// TwinCAT 3 PLC project PersoneelsData
// ProgramVersion: 3.1.4024.0
// libraries:
//   StringUtils, * (System)
//   Tc2_Standard, * (Beckhoff Automation GmbH)
//   Tc2_System, * (Beckhoff Automation GmbH)
//   Tc3_Module, * (Beckhoff Automation GmbH)
// project tree:
//   DUTs/ Pers_data.TcDUT
//   / PlcTask.TcTTO
//   POUs/ FB_CheckString.TcPOU, MAIN.TcPOU
// (motion and I/O tree: see PLC project checkerfunctions)
// real-time tasks:
//   TASK PlcTask: cycle T#10ms, priority 20, ADS port 350
//   TASK PlcTask1: cycle T#10ms, priority 21, ADS port 351
//   TASK PlcTask2: cycle T#10ms, priority 22, ADS port 352
//   TASK PlcTask3: cycle T#10ms, priority 23, ADS port 353
//   TASK PlcTask4: cycle T#10ms, priority 24, ADS port 354
//   TASK PlcTask5: cycle T#10ms, priority 25, ADS port 355
//   TASK PlcTask6: cycle T#10ms, priority 26, ADS port 356
//   TASK PlcTask7: cycle T#10ms, priority 27, ADS port 357

CONFIGURATION PersoneelsData
    RESOURCE PLC ON TwinCAT3
        TASK PlcTask(INTERVAL := T#10ms, PRIORITY := 24);
        PROGRAM MAIN WITH PlcTask : MAIN;
    END_RESOURCE
END_CONFIGURATION

// ---- DUTs/Pers_data.TcDUT
TYPE Pers_data :
STRUCT
    Name : STRING[25];
    Firstname : STRING[25];
    Gender : STRING[10]; // 'Male' of 'Female'
    Age : INT;
    Address : STRING[55];
END_STRUCT
END_TYPE

// ---- POUs/MAIN.TcPOU
PROGRAM MAIN
VAR
    PersonnelArray : ARRAY [1..6] OF Pers_data := [
        (Name := 'Müller', Firstname := 'Peter', Gender := 'Male', Age := 32, Address := 'Postweg 34'),
        (Name := 'Fossen', Firstname := 'Jo', Gender := 'Male', Age := 20, Address := 'Broekstraat 45'),
        (Name := 'Maesen', Firstname := 'Stijn', Gender := 'Male', Age := 15, Address := 'Grote steenweg 8'),
        (Name := 'Poesmans', Firstname := 'Benny', Gender := 'Male', Age := 72, Address := 'Veldweg 1A'),
        (Name := 'Paque', Firstname := 'Stéphanie', Gender := 'Female', Age := 42, Address := 'Tongersesteenweg 456'),
        (Name := 'Dybek', Firstname := 'Isolde', Gender := 'Female', Age := 55, Address := 'Slagerijstraat 6')
    ];
	
	myData : Pers_data; // Vul myData met de gewenste waarden
    searchString : STRING := 'Stijn'; // De te zoeken string
    result : BOOL; // Resultaat van de zoekactie
    checkStringFB : FB_CheckString; // Aanmaken van de FB-instance
END_VAR

// NOG NIET OPGELOST!!!


// Vul myData met gegevens

checkStringFB.data := myData;
checkStringFB.searchString := searchString;

// Roep de FB aan
checkStringFB();

// Haal het resultaat op
result := checkStringFB.found;

END_PROGRAM

// ---- POUs/FB_CheckString.TcPOU
FUNCTION_BLOCK FB_CheckString
VAR_INPUT
    data : Pers_data;
    searchString : STRING; // te zoeken string
END_VAR
VAR_OUTPUT
    found : BOOL;
END_VAR

// NOG NIET OPGELOST!!!

found := (FIND(StrToUpperA(data.Name), StrToUpperA(searchString)) <> 0) OR
         (FIND(StrToUpperA(data.Firstname), StrToUpperA(searchString)) <> 0) OR
         (FIND(StrToUpperA(data.Address), StrToUpperA(searchString)) <> 0);

END_FUNCTION_BLOCK
